// Mitsubishi GX Works2 project: inverter   PLC: Q03UDV

PROGRAM MAIN
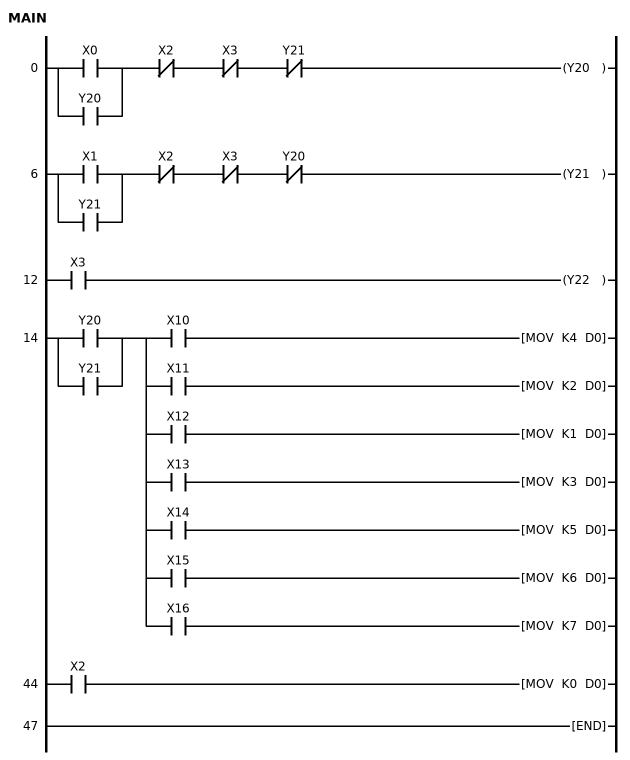
0     LD      X0
      OR      Y20
      ANI     X2
      ANI     X3
      ANI     Y21
      OUT     Y20
6     LD      X1
      OR      Y21
      ANI     X2
      ANI     X3
      ANI     Y20
      OUT     Y21
12    LD      X3
      OUT     Y22
14    LD      Y20
      OR      Y21
      MPS
      AND     X10
      MOV     K4 D0
      MRD
      AND     X11
      MOV     K2 D0
      MRD
      AND     X12
      MOV     K1 D0
      MRD
      AND     X13
      MOV     K3 D0
      MRD
      AND     X14
      MOV     K5 D0
      MRD
      AND     X15
      MOV     K6 D0
      MPP
      AND     X16
      MOV     K7 D0
44    LD      X2
      MOV     K0 D0
47    END
END_PROGRAM

PROGRAM MAIN1
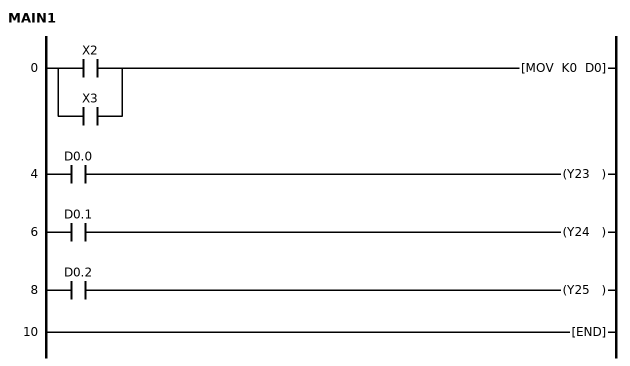
0     LD      X2
      OR      X3
      MOV     K0 D0
4     LD      D0.0
      OUT     Y23
6     LD      D0.1
      OUT     Y24
8     LD      D0.2
      OUT     Y25
10    END
END_PROGRAM
